FUNCTION_BLOCK CompositeFB2
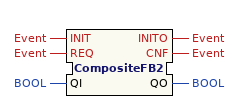
  EVENT_INPUT
    INIT;
    REQ;
  END_EVENT
  EVENT_OUTPUT
    INITO;
    CNF;
  END_EVENT
  VAR_INPUT
    QI : BOOL;
  END_VAR
  VAR_OUTPUT
    QO : BOOL;
  END_VAR
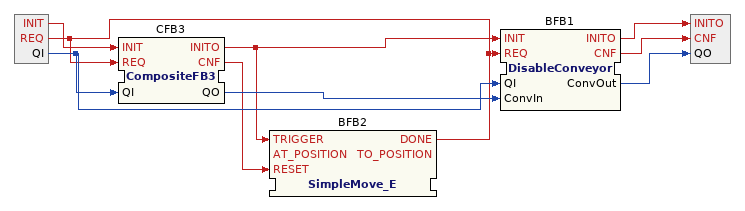
  FBS
    CFB3 : CompositeFB3;
    BFB1 : DisableConveyor;
    BFB2 : SimpleMove_E;
  END_FBS
  EVENT_CONNECTIONS
    INIT TO CFB3.INIT;
    REQ TO CFB3.REQ;
    CFB3.INITO TO BFB1.INIT;
    REQ TO BFB1.REQ;
    CFB3.CNF TO BFB2.RESET;
    BFB2.DONE TO BFB1.REQ;
    CFB3.INITO TO BFB2.TRIGGER;
    BFB1.INITO TO INITO;
    BFB1.CNF TO CNF;
  END_CONNECTIONS
  DATA_CONNECTIONS
    QI TO CFB3.QI;
    BFB1.ConvOut TO QO;
    QI TO BFB1.QI;
    CFB3.QO TO BFB1.ConvIn;
  END_CONNECTIONS
END_FUNCTION_BLOCK
